(* PLC project poST.project, poSTIDE *)
(* stored: creationDateTime 2021-08-31T00:00:00.000000 *)

FUNCTION SUB_TOD_TOD : TIME
  VAR_INPUT
    in1 : TIME_OF_DAY;
    in2 : TIME_OF_DAY;
  END_VAR

END_FUNCTION
